(* IEC 61131-3 sources: eCockpitGit/test_project/src/%F%02 System/%F%03 LoadSaveManager/%POU%FB_LoadSave/%F%Load/%F%Read, 2 files *)

(* ---- %METH%compareString.st ---- *)
//Returns true if the inputted string is the same as the read string
METHOD compareString : BOOL
VAR_INPUT
	str				:POINTER TO EASCII;
END_VAR
(*%!%__DELIMITER__%!%*)
compareString		:=		reader.compareString(str:=str);

(* ---- %METH%readString.st ---- *)
METHOD readString
VAR_INPUT
	str				:POINTER TO EASCII;		//Address of the name to find, only input string address or zero terminated byte array
	lenMax			:DWORD;
END_VAR
VAR_OUTPUT
	len				:WORD;
END_VAR
(*%!%__DELIMITER__%!%*)
reader.readString(str:=str,lenMax:=lenMax,len=>len);
